// TIA Portal V20 export
DATA_BLOCK "LPFE_TelemetryBuffer"   // DB500
// stored: Access Published, MemoryReserve 100, Namespace PFE
   VAR
      buffer { ExternalAccessible := 'False'; ExternalVisible := 'False'; ExternalWritable := 'False'} : Array[0.._.LE_NUMBER_MESSAGES_TELEMETRY_BUFFER] of "LPFE_typePFEDataReqEnvelope250";   // Buffer where record messages are taken from
      mgmtBuffer { ExternalAccessible := 'False'; ExternalVisible := 'False'; ExternalWritable := 'False'} : "LPFE_typeMsgBuffer";   // Mgmt Structure of buffer where record messages are taken from
   END_VAR
BEGIN
END_DATA_BLOCK
